Universal Robots PolyScope program: adam_ur_script.urp

Program adam_ur_script (installation=default directory=/programs/usbdisk createdIn=3.15.8.106339 lastSavedIn=3.15.8.106339 robotSerialNumber=2016331616)
Calibrated DH parameters: a=[-0.000042, -0.244005, -0.113656, 0.000083, 0.000081, 0]; d=[0.152235, -0.912645, 307.527192, -306.50199, 0.085424, 0.082751]; alpha=[1.570617, -0.003934, -0.00059, 1.570394, -1.572717, 0]; deltaTheta=[0.000213, 0.019944, -1.0181, 0.985749, -0.000385, -0.09446]
Robot Program (runOnlyOnce=false)
  Script file /programs/usbdisk/Klientscript1nyeste.script
    | connected = False
    | 
    | while connected == False:
    |      connected = socket_open("192.168.0.5", 30000)  # Forbind til serverens IP-adresse og port
    | end
    | 
    | while (True):
    |     # Send en besked til serveren
    |     socket_send_string("Hello from UR3\n")
    | 
    |     # Modtag en besked fra serveren
    |     response = socket_read_string()
    | 
    |     # Print modtaget besked
    |     textmsg("Received: ", response)
    | 
    |     # Vent et øjeblik før næste iteration
    |     sleep(1.0)
    | 
    | # Luk forbindelsen (dette punkt nås aldrig på grund af den uendelige løkke)
    | socket_close()
    | 
    | end
